# B&R Automation Studio project Khokhlov
Automation Studio 4.5.2.102; Default project

## Configuration Simulation

### Hardware
```
PLC1 : PC_any v1.1.0.0 (OrderNumber=PC)
  VolatileGlobalPvSize = 4096
  XLinkUseDefault = 0
```

## Logical view

Binary libraries used (declarations not repeated): Runtime, Operator, AsIecCon, astime

### Program Logical/Program (ANSIC) - A new program

#### Program.c - Implementation code
```c
/********************************************************************
 * COPYRIGHT --
 ********************************************************************
 * Program: Program
 * File: Program.c
 * Author: admin
 * Created: September 9, 2020
 ********************************************************************
 * Implementation of program Program
 ********************************************************************/

#include <bur/plctypes.h>

#ifdef _DEFAULT_INCLUDES
	#include <AsDefault.h>
#endif

void _INIT ProgramINIT(void)
{
	fb_motor.dt = 0.002;
	fb_motor.ke = 0.00096;
	fb_motor.Tm = 0.04;
	fb_motor.integrator.dt = 0.002;

	fb_motor2.dt = 0.002;
	fb_motor2.ke = 0.00096;
	fb_motor2.Tm = 0.04;
	fb_motor2.integrator.dt = 0.002;

	fb_regulator.dt = 0.002;
	fb_regulator.k_p = 0.0064;
	fb_regulator.k_i = 0.16;
	fb_regulator.max_abs_value = 24;
	fb_regulator.integrator.dt = 0.002;
	enable = 1;
	count = 0;
}

void _CYCLIC ProgramCYCLIC(void)
{
	if(enable)
	{
		count+=10;
		if(count<=2500)
		{
			speed=0;
		}
		else
		{
			speed=6;
			if(count>=5000)
			{
				count=0;
			}
		}
	}
	fb_regulator.e=speed - fb_motor.w;
	fb_motor.u=speed;
	FB_Regulator(&fb_regulator);
	fb_motor.u=fb_regulator.u;
	FB_motor(&fb_motor);

	FB_motor(&fb_motor2);
}
```

#### Program.var - Local variables
```iecst
(********************************************************************
 * COPYRIGHT --
 ********************************************************************
 * Program: Program
 * File: Program.var
 * Author: admin
 * Created: September 9, 2020
 ********************************************************************
 * Local variables of program Program
 ********************************************************************)
VAR
	fb_regulator : FB_Regulator := (0);
	fb_motor : FB_motor := (0);
	speed : REAL := 0.0;
	enable : BOOL := FALSE;
	count : INT := 0;
	fb_motor2 : FB_motor := (0);
END_VAR
```

### Package Logical/Libraries - Global libraries

### Library Logical/Libraries/MtrCtrl (ANSIC) - A new source library

#### MtrCtrl.fun - Exported functions and function blocks
```iecst
(********************************************************************
 * COPYRIGHT --
 ********************************************************************
 * Library: MtrCtrl
 * File: MtrCtrl.fun
 * Author: admin
 * Created: September 9, 2020
 ********************************************************************
 * Functions and function blocks of library MtrCtrl
 ********************************************************************)

FUNCTION_BLOCK FB_Integrator (*TODO: Add your comment here*)
	VAR_INPUT
		in : REAL;
	END_VAR
	VAR_OUTPUT
		out : REAL;
	END_VAR
	VAR
		dt : REAL;
		state : REAL;
	END_VAR
END_FUNCTION_BLOCK

FUNCTION_BLOCK FB_Regulator (*TODO: Add your comment here*)
	VAR_INPUT
		e : REAL;
	END_VAR
	VAR_OUTPUT
		u : REAL;
	END_VAR
	VAR
		k_p : REAL;
		k_i : REAL;
		integrator : FB_Integrator;
		iyOld : REAL;
		max_abs_value : REAL;
		dt : REAL;
	END_VAR
END_FUNCTION_BLOCK

FUNCTION_BLOCK FB_motor (*TODO: Add your comment here*)
	VAR_INPUT
		u : REAL;
	END_VAR
	VAR_OUTPUT
		w : REAL;
		phi : REAL;
	END_VAR
	VAR
		integrator : FB_Integrator;
		Tm : REAL;
		ke : REAL;
		dt : REAL;
	END_VAR
END_FUNCTION_BLOCK
```

#### FB_Integrator.c
```c
/********************************************************************
 * COPYRIGHT --
 ********************************************************************
 * Library: MtrCtrl
 * File: FB_Integrator.c
 * Author: admin
 * Created: September 9, 2020
 ********************************************************************
 * Implementation of library MtrCtrl
 ********************************************************************/

#include <bur/plctypes.h>
#ifdef __cplusplus
	extern "C"
	{
#endif

	#include "MtrCtrl.h"

#ifdef __cplusplus
	};
#endif

/* TODO: Add your comment here */
void FB_Integrator(struct FB_Integrator* inst)
{
	inst->out += inst->in*inst->dt +  inst->state;
	inst->state = inst->out;
	/*TODO: Add your code here*/
}
```

#### FB_Regulator.c
```c
/********************************************************************
 * COPYRIGHT --
 ********************************************************************
 * Library: MtrCtrl
 * File: FB_Regulator.c
 * Author: admin
 * Created: September 9, 2020
 ********************************************************************
 * Implementation of library MtrCtrl
 ********************************************************************/

#include <bur/plctypes.h>
#ifdef __cplusplus
	extern "C"
	{
#endif

	#include "MtrCtrl.h"

#ifdef __cplusplus
	};
#endif

/* TODO: Add your comment here */
void FB_Regulator(struct FB_Regulator* inst)
{
	REAL a = inst->e*inst->k_p;
	REAL b = inst->e*inst->k_i;
	a = a>inst->max_abs_value ? inst->max_abs_value:a;
	a = a<-inst->max_abs_value ? -inst->max_abs_value:a;

	inst->iyOld = inst->integrator.in*b  + inst->iyOld;
	//inst->integrator.in*b + inst->iyOld;
	FB_Integrator(&inst->integrator);
	REAL sum = a + inst->integrator.out;
	inst->u=sum;
	inst->u=inst->u > inst->max_abs_value ? inst->max_abs_value:inst->u;
	inst->u=inst->u < -inst->max_abs_value ? -inst->max_abs_value:inst->u;
	inst->iyOld=inst->u-sum;
}
```

#### FB_Motor.c
```c
/********************************************************************
 * COPYRIGHT --
 ********************************************************************
 * Library: MtrCtrl
 * File: FB_Motor.c
 * Author: admin
 * Created: September 9, 2020
 ********************************************************************
 * Implementation of library MtrCtrl
 ********************************************************************/

#include <bur/plctypes.h>
#ifdef __cplusplus
	extern "C"
	{
#endif

	#include "MtrCtrl.h"

#ifdef __cplusplus
	};
#endif

/* TODO: Add your comment here */
void FB_motor(struct FB_motor* inst)
{
	REAL a = inst->u / inst->ke - inst->w;
	REAL b = a / inst->Tm;
	inst->integrator.in = b;
	FB_Integrator(&inst->integrator);

	inst->w = inst->integrator.out;
	/*TODO: Add your code here*/
}
```
